// TIA Portal V20 export
TYPE "UDT_Flowmeter_Stoe"
   STRUCT
      "No Flow Detected" : Bool;   // No liquid is flowing through the sensor.
      "Flow Rate Too Low" : Bool;   // The measured flow is below the minimum threshold.
      "Flow Rate Too Hight" : Bool;   // The measured flow exceeds the maximum allowed value.
      "Sensor CH1_wBreak" : Bool;   // The flow sensor CH1 is not connected or has a broken wire
      "Sensor CH2_wBreak" : Bool;   // The flow sensor CH2 is not connected or has a broken wire
      "Temprature Above Limit" : Bool;
      "Flow Out Of Range" : Bool;   // The sensor output signal is outside the valid range (e.g. 0–10 V or 4–20 mA)
      "Calibration Error" : Bool;   // The flow sensor is not calibrated correctly
      "Air Bubles Detected" : Bool;   // Air bubbles in the liquid are affecting the flow measurement
      "Temprature Out Of Range" : Bool;   // Liquid temperature is outside the sensor’s operating range
      "Temprature Below Limit" : Bool;
      "Reverse Flow Detected" : Bool;   // Flow is moving in the opposite direction
      "Communcation Error" : Bool;   // No communication between sensor and controller (PLC)
      "Clogging or Blockage" : Bool;   // The flow path is blocked or partially obstructed
      "Sensor Overheating" : Bool;   // The sensor temperature is too high
      "Dirty Sensor" : Bool;   // Deposits or dirt on the sensor are affecting measurement accuracy
   END_STRUCT;
END_TYPE
